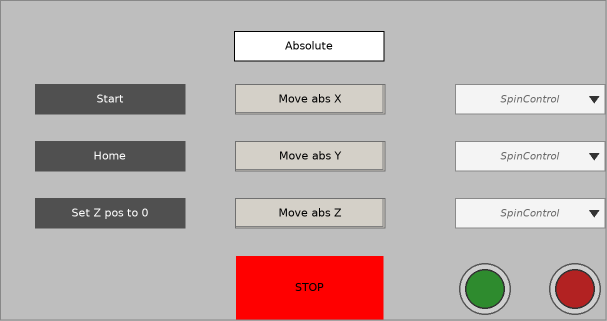
VISUALIZATION goPositionAbs  // 607x321
    Button (235,84 150x30), "Move abs X"
        tap POSITION.DoAbs_X
    Button (235,141 150x30), "Move abs Y"
        tap POSITION.DoAbs_Y
    Button (235,198 150x30), "Move abs Z"
        tap POSITION.DoAbs_Z
    Rectangle (35,141 150x30), "Home"
        tap INIT.bHome
    Rectangle (35,84 150x30), "Start", colour toggle: INIT.bENCouple
        toggle INIT.bENCouple
    Rectangle (35,198 150x30), "Set Z pos to 0"
        tap POSITION.SetZpos
    SpinControl (455,84 150x30), variable: POSITION.abs_X
        OnMouseDown: write POSITION.abs_X via Edit, min 0, max 275
    SpinControl (455,141 150x30), variable: POSITION.abs_Y
        OnMouseDown: write POSITION.abs_Y via Edit, min 0, max 275
    SpinControl (455,198 150x30), variable: POSITION.abs_Z
        OnMouseDown: write POSITION.abs_Z via Edit, min 0, max 90
    Rectangle (236,256 147x63), "STOP", colour toggle: GVL.StopALL
        toggle GVL.StopALL
    Lamp1 (455,259 60x60), variable: POSITION.Done, style: Lamp-Lamp1-Green
    Lamp1 (545,259 60x60), variable: POSITION.Busy, style: Lamp-Lamp1-Red
    Rectangle (234,31 150x30), "Absolute"
END_VISUALIZATION

(* stored: Version 1.1.0.1, ProductVersion 3.1.4022.17
   Visu goPositionAbs: Id {0a2c3fad-856f-4a03-964e-a4d38d5333e4} *)
